Staubli VAL3: onEnterEvent.pgx

program onEnterEvent(string x_sName, bool& x_bSave[])
  local num i
  local string l_sProg
  local num l_nIndex
  local point l_pPoint[2]
  local string l_sEmpty
  local TrajPallet l_tPallet
  local num l_nPos
  local num l_nSize
  local num l_nXYZ[3]
  local num z
  local num y
  local num x
  local num l_nX
  local num l_nY
  local num l_nZ
  local num j
  local num l_nId
begin
  //
  // NB sEvent is the selected
  // element in the LIST
  //
  if nIndex>=0
    call use:findPos(sEvent,">",i)
    i=i+1
  endIf
  //
  // update all the value
  //
  call pallet:getSizeItem(false,l_nSize)
  call pallet:getPalletData(false,l_tPallet)
  call pallet:getPalletPos(x_sName,l_nPos)
  // make the default
  if l_nSize>=1
    // ORIGIN
    call pallet:getPoint(l_pPoint,false,0)

    fFather=tTrajPallet.fReference
    pO.trsf=position(l_pPoint,fFather)
    pOrigin.trsf=position(pO,l_tPallet.fFrame)
  endIf
  // clean the line
  call use:listcursor(use:nView,false)
  // swith the line
  // use this
  // l_nPos=(nX*nY)*(l_nZ-1)+(nX)*(l_nY-1)+(l_nX-1))
  // call setPalletPos(x_sItem,(l_nSize[0]*l_nSize[2])*(l_nValue[3]-1)+(l_nSize[0])*(l_nValue[2]-1)+(l_nValue[1]-1))
  l_nX=(l_nPos%(l_tPallet.nX*l_tPallet.nY))%l_tPallet.nX+1
  l_nY=roundDown((l_nPos%(l_tPallet.nX*l_tPallet.nY))/l_tPallet.nX)+1
  l_nZ=roundDown(l_nPos/(l_tPallet.nX*l_tPallet.nY))+1
  switch nIndex
    case 0
      // absolute
      l_sEmpty=""
      l_nPos=l_nPos+1
      call use:changeValue(l_nPos,1,l_nSize,i+40-use:nBottomX,use:nView+1,l_sEmpty)
      call pallet:setPalletPos(x_sName,l_nPos-1)
    break
    case 1
      // X value
      l_sEmpty=""
      call use:changeValue(l_nX,1,l_tPallet.nX,i+40-use:nBottomX,use:nView+1,l_sEmpty)
    break
    case 2
      // Y value
      l_sEmpty=""
      call use:changeValue(l_nY,1,l_tPallet.nY,i+40-use:nBottomX,use:nView+1,l_sEmpty)
    break
    case 3
      // Z value
      l_sEmpty=""
      call use:changeValue(l_nZ,1,l_tPallet.nZ,i+40-use:nBottomX,use:nView+1,l_sEmpty)
    break
    case 4,5,6
      // dx dy dz
      if l_nSize>1
        //get the old one
        for j=0 to 2
          l_nXYZ[j]=l_tPallet.nDistanceXYZ[j]
        endFor
        call use:changeValue(l_tPallet.nDistanceXYZ[nIndex-4],0,0,i+40-use:nBottomX,use:nView+1,l_sEmpty)
        // update it
        call pallet:setPalletData(l_tPallet)
        // set the offset
        l_nXYZ[0]=l_tPallet.nDistanceXYZ[0]-l_nXYZ[0]
        l_nXYZ[1]=l_tPallet.nDistanceXYZ[1]-l_nXYZ[1]
        l_nXYZ[2]=l_tPallet.nDistanceXYZ[2]-l_nXYZ[2]
        // change the offset for all
        call pallet:changeOffset(l_nXYZ)
        // update the value back
        call pallet:getPalletData(false,l_tPallet)
        use:bUseRefresh=true
        x_bSave=true
      endIf
    break
    //
    default
      // plane line action
      if nIndex>=7
        l_nIndex=nIndex-7
        l_sProg=right(sEvent,len(sEvent)-i)
        call programList(l_sProg)
        l_tPallet.sAction[l_nIndex]=l_sProg
        x_bSave=true
      endIf
    break
  endSwitch
  // update the position
  if nIndex>=1 and nIndex<=3
    l_nPos=(l_tPallet.nX*l_tPallet.nY)*(l_nZ-1)+(l_tPallet.nX)*(l_nY-1)+(l_nX-1)
    call pallet:setPalletPos(x_sName,l_nPos)
  endIf
  // update all
  if x_bSave
    call pallet:setPalletData(l_tPallet)
    call pallet:getPalletData(false,tTrajPallet)
  endIf
  // refresh it
  call buildList()
  use:bUseRefresh=true
end
